(* CODESYS project Lyntupy.project
   Title: Lypuny
   Author: d2581
   Version: 0.0.0.92

Project tree, tasks and I/O mapping:
  MyController : TM241CE40T/U, Schneider Electric, order no. TM241CE40T/U, version 4.0.6.18
    application Application
      libraries: Util, 3.5.1.0 (System)
      task MAST (cyclic, interval 20 ms, priority 15, watchdog 100 ms x 1) calls FirstMastCycle, Input, PumpsFeederWater, AnalogInput, MeteoVlvPid, VlvRezervTankWtr, SetResetErr, FactorySetup, PumpsSourceWater, PumpsNetWater, Output
      global variables GVL
      global variables GVL_RETAIN
      FB/
        function block InitializationTmpGrafik [ST]
        function block OutputLimit [ST]
        function block ControlMeteoVlv [ST]
        function block ControlMeteoValve [FBD]
        function block DerjatelTemperatury [ST]
        function block OpredelaetPosition [LD]
        function block regulirovshchyk_rejyma [LD]
      PRG/
        program Input [ST]
        program Output [ST]
        program PumpsNetWater [LD]
        program PumpsFeederWater [LD]
        program PumpsSourceWater [LD]
        program VlvRezervTankWtr [LD]
        program MeteoVlvPid [FBD]
        program AnalogInput [FBD]
        program SetResetErr [LD]
        program FactorySetup [LD]
        program FirstMastCycle [CFC]
      VAR/
      global variables SystemBit
      function CheckDivDInt [ST]
      function CheckDivLInt [ST]
      function CheckDivReal [ST]
      function CheckDivLReal [ST]
    A1_IN : Digital Inputs, Schneider Electric, version 4.0.6.18
        input  idwDI_IDW0 : DWORD  // IDW0
        input  X0 : BOOL  // IDW0.I0
        input  X1 : BOOL  // IDW0.I1
        input  X2 : BOOL  // IDW0.I2
        input  X3 : BOOL  // IDW0.I3
        input  X4 : BOOL  // IDW0.I4
        input  X5 : BOOL  // IDW0.I5
        input  X6 : BOOL  // IDW0.I6
        input  X7 : BOOL  // IDW0.I7
        input  X8 : BOOL  // IDW0.I8
        input  X9 : BOOL  // IDW0.I9
        input  X10 : BOOL  // IDW0.I10
        input  X11 : BOOL  // IDW0.I11
        input  X12 : BOOL  // IDW0.I12
        input  X13 : BOOL  // IDW0.I13
        input  X14 : BOOL  // IDW0.I14
        input  X15 : BOOL  // IDW0.I15
        input  X16 : BOOL  // IDW0.I16
        input  X17 : BOOL  // IDW0.I17
        input  X18 : BOOL  // IDW0.I18
        input  X19 : BOOL  // IDW0.I19
        input  X20 : BOOL  // IDW0.I20
        input  X21 : BOOL  // IDW0.I21
        input  X22 : BOOL  // IDW0.I22
        input  X23 : BOOL  // IDW0.I23
        input  ibDI_IB1 : BYTE  // IB1
    A1_OUT : Digital Outputs, Schneider Electric, version 4.0.6.18
        output Y0 : BOOL  // QW0.Q0
        output Y1 : BOOL  // QW0.Q1
        output Y2 : BOOL  // QW0.Q2
        output Y3 : BOOL  // QW0.Q3
        output Y4 : BOOL  // QW0.Q4
        output Y5 : BOOL  // QW0.Q5
        output Y6 : BOOL  // QW0.Q6
        output Y7 : BOOL  // QW0.Q7
        output Y8 : BOOL  // QW0.Q8
        output Y9 : BOOL  // QW0.Q9
        output Y10 : BOOL  // QW0.Q10
        output Y11 : BOOL  // QW0.Q11
        output Y12 : BOOL  // QW0.Q12
        output Y13 : BOOL  // QW0.Q13
        output Y14 : BOOL  // QW0.Q14
        output Y15 : BOOL  // QW0.Q15
        output qbDQ_QB1 : BYTE  // QB1
        unmapped channels: QW0
    Counters : Counters, Schneider Electric, version 4.0.6.18
    Pulse_Generators : Pulse Generators, Schneider Electric, version 4.0.6.18
    Cartridge_1 : Cartridge, Schneider Electric, version 4.0.6.18
    Cartridge_2 : Cartridge, Schneider Electric, version 4.0.6.18
    IO_Bus : IO bus - TM3, Schneider Electric, version 4.0.6.18
      A1_1 : TM3DI16K, Schneider Electric, order no. TM3DI16K, version 1.0.1.4
          input  iwModule_1_IW0 : WORD  // IW0
          input  _1X0 : BOOL  // IW0.I0
          input  _1X1 : BOOL  // IW0.I1
          input  _1X2 : BOOL  // IW0.I2
          input  _1X3 : BOOL  // IW0.I3
          input  _1X4 : BOOL  // IW0.I4
          input  _1X5 : BOOL  // IW0.I5
          input  _1X6 : BOOL  // IW0.I6
          input  _1X7 : BOOL  // IW0.I7
          input  _1X8 : BOOL  // IW0.I8
          input  _1X9 : BOOL  // IW0.I9
          input  _1X10 : BOOL  // IW0.I10
          input  _1X11 : BOOL  // IW0.I11
          input  _1X12 : BOOL  // IW0.I12
          input  _1X13 : BOOL  // IW0.I13
          input  _1X14 : BOOL  // IW0.I14
          input  _1X15 : BOOL  // IW0.I15
      A1_2 : TM3DQ16TK, Schneider Electric, order no. TM3DQ16TK, version 1.0.1.4
          output _2Y0 : BOOL  // QW0.Q0
          output _2Y1 : BOOL  // QW0.Q1
          output _2Y2 : BOOL  // QW0.Q2
          output _2Y3 : BOOL  // QW0.Q3
          output _2Y4 : BOOL  // QW0.Q4
          output _2Y5 : BOOL  // QW0.Q5
          output _2Y6 : BOOL  // QW0.Q6
          output _2Y7 : BOOL  // QW0.Q7
          output _2Y8 : BOOL  // QW0.Q8
          output _2Y9 : BOOL  // QW0.Q9
          output _2Y10 : BOOL  // QW0.Q10
          output _2Y11 : BOOL  // QW0.Q11
          output _2Y12 : BOOL  // QW0.Q12
          output _2Y13 : BOOL  // QW0.Q13
          output _2Y14 : BOOL  // QW0.Q14
          output _2Y15 : BOOL  // QW0.Q15
          unmapped channels: QW0
      A1_3 : TM3AI4/G, Schneider Electric, order no. TM3AI4/G, version 1.0.0.15
          settings: KPI Configuration.KPI Configuration[0] = 35; KPI Configuration.KPI Configuration[1] = 35; KPI Configuration.KPI Configuration[2] = 35; KPI Configuration.KPI Configuration[3] = 35; KPI Configuration.KPI Configuration[4] = 160; KPI Configuration.KPI Configuration[5] = 15; KPI Configuration.KPI Configuration[6] = 160; KPI Configuration.KPI Configuration[7] = 15; KPI Configuration.KPI Configuration[8] = 160; KPI Configuration.KPI Configuration[9] = 15; KPI Configuration.KPI Configuration[10] = 160; KPI Configuration.KPI Configuration[11] = 15; KPI Configuration.KPI Configuration[12] = 32; KPI Configuration.KPI Configuration[13] = 78; KPI Configuration.KPI Configuration[14] = 32; KPI Configuration.KPI Configuration[15] = 78; KPI Configuration.KPI Configuration[16] = 32; KPI Configuration.KPI Configuration[17] = 78; KPI Configuration.KPI Configuration[18] = 32; KPI Configuration.KPI Configuration[19] = 78; KPI Configuration.KPI Configuration[20] = 1; KPI Configuration.KPI Configuration[22] = 1; KPI Configuration.KPI Configuration[24] = 1; KPI Configuration.KPI Configuration[26] = 1; KPI Configuration.KPI Configuration[29] = 1; KPI Configuration.KPI Configuration[30] = 1; KPI Configuration.KPI Configuration[31] = 1
          input  PE1 : INT  // IW0
          input  PE2 : INT  // IW1
          input  PE3 : INT  // IW2
          input  PERezerv : INT  // IW3
          input  ibModule_3_IBStatusIW0 : BYTE  // IBStatusIW0
          input  ibModule_3_IBStatusIW1 : BYTE  // IBStatusIW1
          input  ibModule_3_IBStatusIW2 : BYTE  // IBStatusIW2
          input  ibModule_3_IBStatusIW3 : BYTE  // IBStatusIW3
      A1_4 : TM3TI4/G, Schneider Electric, order no. TM3TI4/G, version 1.0.1.5
          settings: KPI Configuration.KPI Configuration[0] = 77; KPI Configuration.KPI Configuration[1] = 77; KPI Configuration.KPI Configuration[2] = 77; KPI Configuration.KPI Configuration[3] = 77; KPI Configuration.KPI Configuration[4] = 48; KPI Configuration.KPI Configuration[5] = 248; KPI Configuration.KPI Configuration[6] = 48; KPI Configuration.KPI Configuration[7] = 248; KPI Configuration.KPI Configuration[8] = 48; KPI Configuration.KPI Configuration[9] = 248; KPI Configuration.KPI Configuration[10] = 48; KPI Configuration.KPI Configuration[11] = 248; KPI Configuration.KPI Configuration[12] = 52; KPI Configuration.KPI Configuration[13] = 33; KPI Configuration.KPI Configuration[14] = 52; KPI Configuration.KPI Configuration[15] = 33; KPI Configuration.KPI Configuration[16] = 52; KPI Configuration.KPI Configuration[17] = 33; KPI Configuration.KPI Configuration[18] = 52; KPI Configuration.KPI Configuration[19] = 33; KPI Configuration.KPI Configuration[20] = 1; KPI Configuration.KPI Configuration[22] = 1; KPI Configuration.KPI Configuration[26] = 1
          input  TE1 : INT  // IW0
          input  TE2 : INT  // IW1
          input  TE3 : INT  // IW2
          input  TE4Rezerv : INT  // IW3
          input  ibModule_4_IBStatusIW0 : BYTE  // IBStatusIW0
          input  ibModule_4_IBStatusIW1 : BYTE  // IBStatusIW1
          input  ibModule_4_IBStatusIW2 : BYTE  // IBStatusIW2
          input  ibModule_4_IBStatusIW3 : BYTE  // IBStatusIW3
    COM_Bus : COM bus, Schneider Electric, version 4.0.6.18
    Ethernet_1 : Ethernet Network, Schneider Electric, version 4.0.6.18
        settings: IPAddress = [192, 168, 0, 32]; SubnetMask = [255, 255, 255, 0]; WebServer = TRUE; FTP Server = TRUE; SoMachine Protocol = TRUE; Modbus Server = TRUE; NetManage Protocol = TRUE; SNMP protocol = TRUE; Enable Routing = FALSE; WebVisu protocol = TRUE; DHCP Server Active = TRUE
    Serial_Line_1 : Serial line, Schneider Electric, version 4.0.6.18
      Modbus_Manager : Modbus Manager, Schneider Electric, version 4.0.0.2
    Serial_Line_2 : Serial line, Schneider Electric, version 4.0.6.18
*)

// MyController/Application/GVL
VAR_GLOBAL
	//------------------------------------------------------Inpup A1 A1.1 A1.3 A1.4-----------------------------------------
	Breake1 AT %MX0.0: BOOL;
	ErrBoiler1 AT %MX0.1: BOOL;
	ManualMode AT %MX0.2: BOOL;
	ErrBoiler2 AT %MX0.3: BOOL;
	Breake2 AT %MX0.4: BOOL;
	PressReversNetWtrLow AT %MX0.5: BOOL;
	PressReversNetWtrHigh AT %MX0.6: BOOL;
	DrySourceWtr1 AT %MX0.7: BOOL;
	WorkingPressSourceWtr1 AT %MX0.8: BOOL;
	DrySourceWtr2 AT %MX0.9: BOOL;
	WorkingPressSourceWtr2 AT %MX0.10: BOOL;
	DryNetWtr1 AT %MX0.11: BOOL;
	WorkingPressNetWtr1 AT %MX0.12: BOOL;
	DryNetWtr2 AT %MX0.13: BOOL;
	WorkingPressNetWtr2 AT %MX0.14: BOOL;
	DryFeederWtr1 AT %MX0.15: BOOL;
	WorkingPressFeederWtr1 AT %MX2.0: BOOL;
	DryFeederWtr2 AT %MX2.1: BOOL;//%MW1.1
	WorkingPressFeederWtr2 AT %MX2.2: BOOL;//%MW1.2
	PumpSourceWtr1On AT %MX2.3: BOOL;//%MW1.3
	PumpSourceWtr2On AT %MX2.4: BOOL;//%MW1.4
	PumpNetWtr1On AT %MX2.5: BOOL;//%MW1.5
	PumpNetWtr2On AT %MX2.6: BOOL;//%MW1.6
	PumpFeederWtr1On AT %MX2.7: BOOL;//%MW1.7
	PumpFeederWtr2On AT %MX2.8: BOOL;//%MW1.8
	ErrTopLevelReservTankWtr AT %MX2.9: BOOL;//%MW1.9
	TopLevelReservTankWtr AT %MX2.10: BOOL;//%MW1.10
	ErrLowLevelReservTankWtr AT %MX2.11: BOOL;//%MW1.11
	LowLevelReservTankWtr AT %MX2.12: BOOL;//%MW1.12
	Breake3 AT %MX2.13: BOOL;//%MW1.13
	// --------------------------------------------------------------резервные биты в слове -----------------------------------------------
	ErrGrafik AT %MX2.14: BOOL;
	ErrPE1 AT %MX2.15: BOOL;
	// -------------------------------------------------------------------------------------------------------------------------------------
	PressReversNetWtr AT %MD1: REAL;//%MW2,%MW3
	PressForwardNetWtr AT %MD3: REAL;//%MW6,%MW7
	PressSourceWtr AT %MD5: REAL;//%MW10,%MW11
	TpmReversNetWtr AT %MW14: INT;
	TmpAir AT %MW15: INT;
	TmpForwardWtr AT %MW16: INT;
	//------------------------------------------------------Outpun A1------------------------------------------------
	ErrPE2 AT %MX34.0: BOOL;//%MW17:X0 в панели
	PumpNetWtr1Run AT %MX34.1: BOOL;
	PumpNetWtr1Stop AT %MX34.2: BOOL;
	PumpNetWtr2Run AT %MX34.3: BOOL;
	PumpNetWtr2Stop AT %MX34.4: BOOL;
	PumpFeeder1Run AT %MX34.5: BOOL;
	PumpFeeder1Stop AT %MX34.6: BOOL;
	PumpFeeder2Run AT %MX34.7: BOOL;
	PumpFeeder2Stop AT %MX34.8: BOOL;
	PumpSourceWtr1Run AT %MX34.9: BOOL;
	PumpSourceWtr1Stop AT %MX34.10: BOOL;
	PumpSourceWtr2Run AT %MX34.11: BOOL;
	PumpSourceWtr2Stop AT %MX34.12: BOOL;
	VlvRezervTankWtrOpen AT %MX34.13: BOOL;
	RezervY13 AT %MX34.14: BOOL;
	VlvBypassOpen AT %MX34.15: BOOL;
	VlvBypassClose AT %MX36.0: BOOL;
	LightSignalColumn AT %MX36.1: BOOL;
	// --------------------------------------------------3 реле в резерве-----------------------------------------------
	Rezerv2Y1 AT %MX36.2: BOOL;
	Rezerv2Y2 AT %MX36.3: BOOL;
	Rezerv2Y3 AT %MX36.4: BOOL;
	// --------------------------------------------------резервные биты в слове-----------------------------------------
	ErrPE3 AT %MX36.5: BOOL;
	ErrTE1 AT %MX36.6: BOOL;
	ErrTE2 AT %MX36.7: BOOL;
	ErrTE3 AT %MX36.8: BOOL;
	BtnResetErr AT %MX36.9: BOOL;
	HandModeMeteo AT %MX36.10: BOOL;
	BtnRunOpnMeteoVlv AT %MX36.11: BOOL;
	BtnRunClsMeteoVlv AT %MX36.12: BOOL;
	BtnRunPumpFeederWtr1 AT %MX36.13: BOOL;
	BtnRunPumpFeederWtr2 AT %MX36.14: BOOL;
	BtnRunPumpNetWtr1 AT %MX36.15: BOOL;
	// -----------------------------------------------------------------------------------------------------------------
	BtnRunPumpNetWtr2 AT %MX80.0: BOOL;//%MW40:X0 в панели
	BtnRunPumpSourceWtr1 AT %MX80.1: BOOL;
	BtnRunPumpSourceWtr2 AT %MX80.2: BOOL;
	BtnVlvRezervTankWtrOpen AT %MX80.3: BOOL;//%MW40:X3
	ErrAll AT %MX80.4: BOOL;//%MW40:X4
	BtnSetFactorySetup AT %MX80.5: BOOL;//%MW40:X5
	bool6 AT %MX80.6: BOOL;//%MW40:X6
	bool7 AT %MX80.7: BOOL;//%MW40:X7
	bool8 AT %MX80.8: BOOL;//%MW40:X8
	bool9 AT %MX80.9: BOOL;//%MW40:X9
	bool10 AT %MX80.10: BOOL;//%MW40:X10
	bool11 AT %MX80.11: BOOL;//%MW40:X11
	bool12 AT %MX80.12: BOOL;//%MW40:X12
	bool13 AT %MX80.13: BOOL;//%MW40:X13
	bool14 AT %MX80.14: BOOL;//%MW40:X14
	bool15 AT %MX80.15: BOOL;//%MW40:X15
	
	LevelRezervTankWtr AT %MW41: INT;
	ZadanieForMeteoVlv AT %MW42: INT;

END_VAR

// MyController/Application/GVL_RETAIN
VAR_GLOBAL RETAIN
	PE1Min AT %MW4: INT;
	PE1Max AT %MW5: INT;
	PE2Min AT %MW8: INT;
	PE2Max AT %MW9: INT;
	PE3Min AT %MW12: INT;
	PE3Max AT %MW13: INT;
	
	
	TmpGrafN22 AT %MW19: WORD;
	TmpGrafN19 AT %MW20: WORD;
	TmpGrafN15 AT %MW21: WORD;
	TmpGrafN13 AT %MW22: WORD;
	TmpGrafN10 AT %MW23: WORD;
	TmpGrafN7 AT %MW24: WORD;
	TmpGrafN3 AT %MW25: WORD;
	TmpGrafP0 AT %MW26: WORD;
	TmpGrafP2 AT %MW27: WORD;
	TmpGrafP5 AT %MW28: WORD;
	TmpgrafP10 AT %MW29: WORD;
	
	KL: ARRAY[0..10] OF POINT;
	
	KpVlv AT %MD15: REAL;// %MW30, %MW31
	TnVlv AT %MD16: REAL;// %MW32, %MW33
	TvVlv AT %MD17: REAL;// %MW34, %MW35
	MaxVlv AT %MW36: INT;//Максимальная величина открытия задвижки в %
	MinVlv AT %MW37: INT;//Минимальная величина закрытия задвижки в %
	TimeMoveVlv AT %MW38: INT;//Время открытия задвижки в секундах
	CurrentPositionVlv AT %MW39: INT;// Текущее положение
	
	UseM1 AT %MX86.0: BOOL;
	UseM2 AT %MX86.1: BOOL;
	UseM3 AT %MX86.2: BOOL;
	UseM4 AT %MX86.3: BOOL;
	UseM5 AT %MX86.4: BOOL;
	UseM6 AT %MX86.5: BOOL;
	
	CurrentPosition: INT;
END_VAR

// MyController/Application/SystemBit
VAR_GLOBAL
	// Indicates or executes a cold start (data initialized to default values)
	SB_COLDSTART: BOOL;
	// Indicates there was a warm start with data backup
	SB_WARMSTART: BOOL;
	// Time base of 1 min generated by an internal clock
	SB_TB1MIN: BOOL;
	// Time base of 1 sek generated by an internal clock
	SB_TB1SEK: BOOL;
	// Indicates the first controller cycle in RUN mode
	SB_FIRSTRUN: BOOL;
END_VAR

// MyController/Application/PRG/FirstMastCycle
PROGRAM FirstMastCycle
VAR
	tm_firstrun: TOF;
	BLINK_1sek: Util.BLINK;
END_VAR
VAR // added by the converter: edge detectors and wires of the graphical bodies
    _w1 : ANY;
END_VAR

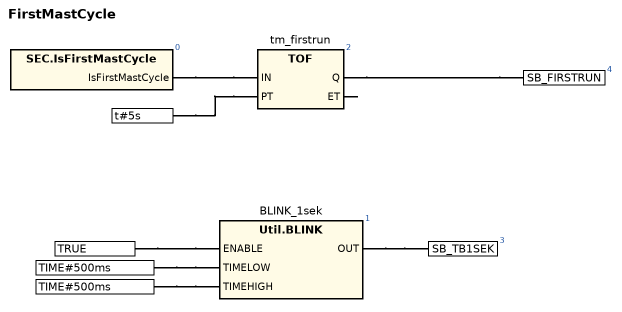
_w1 := SEC.IsFirstMastCycle();
BLINK_1sek(ENABLE := TRUE, TIMELOW := TIME#500ms, TIMEHIGH := TIME#500ms); // Util.BLINK
tm_firstrun(IN := _w1, PT := t#5s); // TOF
SB_TB1SEK := BLINK_1sek.OUT;
SB_FIRSTRUN := tm_firstrun.Q;

END_PROGRAM

// MyController/Application/PRG/Input
PROGRAM Input
VAR
END_VAR

Breake1 := 	NOT X0;
ErrBoiler1 := X1;
ManualMode := X2;
ErrBoiler2 := X3;
Breake2 := X4;
PressReversNetWtrLow := NOT X5;//PIS9
PressReversNetWtrHigh := NOT X6;//PIS9
DrySourceWtr1 := NOT X7;//PIS7
WorkingPressSourceWtr1:= NOT X8;//PIS5
DrySourceWtr2 := NOT X9;//PIS8
WorkingPressSourceWtr2 := NOT X10;//PIS6
DryNetWtr1 := NOT X11;//PIS3
WorkingPressNetWtr1 := NOT X12;//PIS1
DryNetWtr2 := NOT X13;//PIS4
WorkingPressNetWtr2 := NOT X14;//PIS2
DryFeederWtr1 := NOT X15;//PIS11
WorkingPressFeederWtr1 := NOT X16; //PIS9
DryFeederWtr2 := NOT X17;//PIS12
WorkingPressFeederWtr2 := NOT X18; //PIS12
PumpSourceWtr1On := X19;//KM-K6.1
PumpSourceWtr2On := X20;//KM-K6.2
PumpNetWtr1On := X21;//KM-K3.1
PumpNetWtr2On := X22;//KM-K3.2
PumpFeederWtr1On :=	X23;//KM-K4.1
PumpFeederWtr2On := _1X0;//KM-K4.2
ErrTopLevelReservTankWtr := _1X4;//Верхний аварийный уровень в баке запаса воды
TopLevelReservTankWtr := _1X3;//Верхний рабочий уровень в баке запаса воды
ErrLowLevelReservTankWtr := _1X1;//Нижний аварийный уровень в баке запаса воды
LowLevelReservTankWtr := _1X2;//Нижний рабочий уровень в баке запаса воды
Breake3 := _1X5;

PressReversNetWtr := AnalogInput.LinTrafoPressReversNetWtr.OUT;//Давление обратной сетевой воды
PressForwardNetWtr := AnalogInput.LinTrafoPressForwardNetWtr.OUT;//Давление прямой сетевой воды 
PressSourceWtr := AnalogInput.LinTrafoPressSourceWtr.OUT;;//Давление исходной сетевой воды 

TpmReversNetWtr := TE1;//Температура обратной сетевой воды на входе в котельную
TmpForwardWtr := TE2;//Температура прямой сетевой воды на выходе из котельной
TmpAir := TE3;//Температура наружнего воздуха

END_PROGRAM

// MyController/Application/PRG/AnalogInput
PROGRAM AnalogInput
VAR
	LinTrafoPressReversNetWtr: LIN_TRAFO;
	LinTrafoPressForwardNetWtr: LIN_TRAFO;
	LinTrafoPressSourceWtr: LIN_TRAFO;
	ErrPE1: BOOL;
	ErrPE2: BOOL;
	ErrPE3: BOOL;
END_VAR

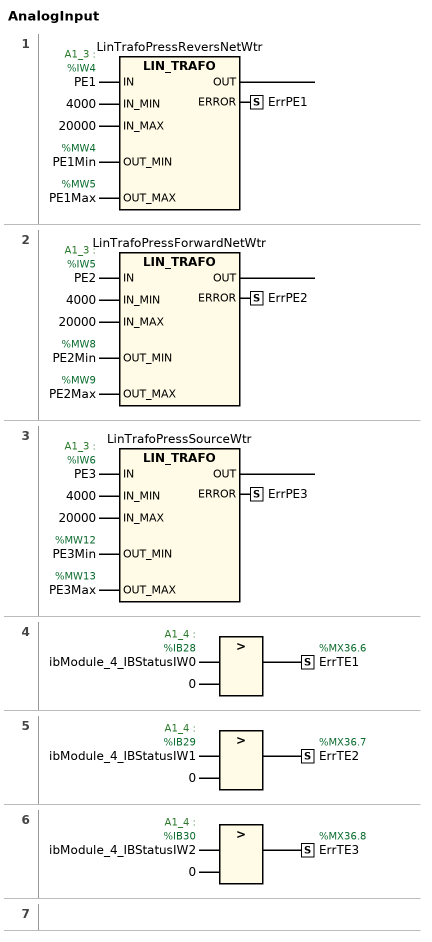
// NETWORK 1
//   PE1: A1_3 : | AT %IW4
//   PE1Min: AT %MW4
//   PE1Max: AT %MW5
LinTrafoPressReversNetWtr(IN := PE1, IN_MIN := 4000, IN_MAX := 20000, OUT_MIN := PE1Min, OUT_MAX := PE1Max); // LIN_TRAFO
ErrPE1 S= LinTrafoPressReversNetWtr.ERROR;

// NETWORK 2
//   PE2: A1_3 : | AT %IW5
//   PE2Min: AT %MW8
//   PE2Max: AT %MW9
LinTrafoPressForwardNetWtr(IN := PE2, IN_MIN := 4000, IN_MAX := 20000, OUT_MIN := PE2Min, OUT_MAX := PE2Max); // LIN_TRAFO
ErrPE2 S= LinTrafoPressForwardNetWtr.ERROR;

// NETWORK 3
//   PE3: A1_3 : | AT %IW6
//   PE3Min: AT %MW12
//   PE3Max: AT %MW13
LinTrafoPressSourceWtr(IN := PE3, IN_MIN := 4000, IN_MAX := 20000, OUT_MIN := PE3Min, OUT_MAX := PE3Max); // LIN_TRAFO
ErrPE3 S= LinTrafoPressSourceWtr.ERROR;

// NETWORK 4
//   ibModule_4_IBStatusIW0: A1_4 : | AT %IB28
//   ErrTE1: AT %MX36.6
ErrTE1 S= ibModule_4_IBStatusIW0 > 0;

// NETWORK 5
//   ibModule_4_IBStatusIW1: A1_4 : | AT %IB29
//   ErrTE2: AT %MX36.7
ErrTE2 S= ibModule_4_IBStatusIW1 > 0;

// NETWORK 6
//   ibModule_4_IBStatusIW2: A1_4 : | AT %IB30
//   ErrTE3: AT %MX36.8
ErrTE3 S= ibModule_4_IBStatusIW2 > 0;

// NETWORK 7

END_PROGRAM

// MyController/Application/PRG/PumpsFeederWater
PROGRAM PumpsFeederWater
VAR
	PulsRunPumpFeederWtr1: TP;
	PulsStopPumpFeederWtr1: TP;
	PulsStopPumpFeederWtr2: TP;
	PulsRunPumpFeederWtr2: TP;
END_VAR
VAR // added by the converter: edge detectors and wires of the graphical bodies
    _w1 : BOOL;
    _rt1, _rt2, _rt3, _rt4 : R_TRIG;
    _ft1, _ft2 : F_TRIG;
END_VAR

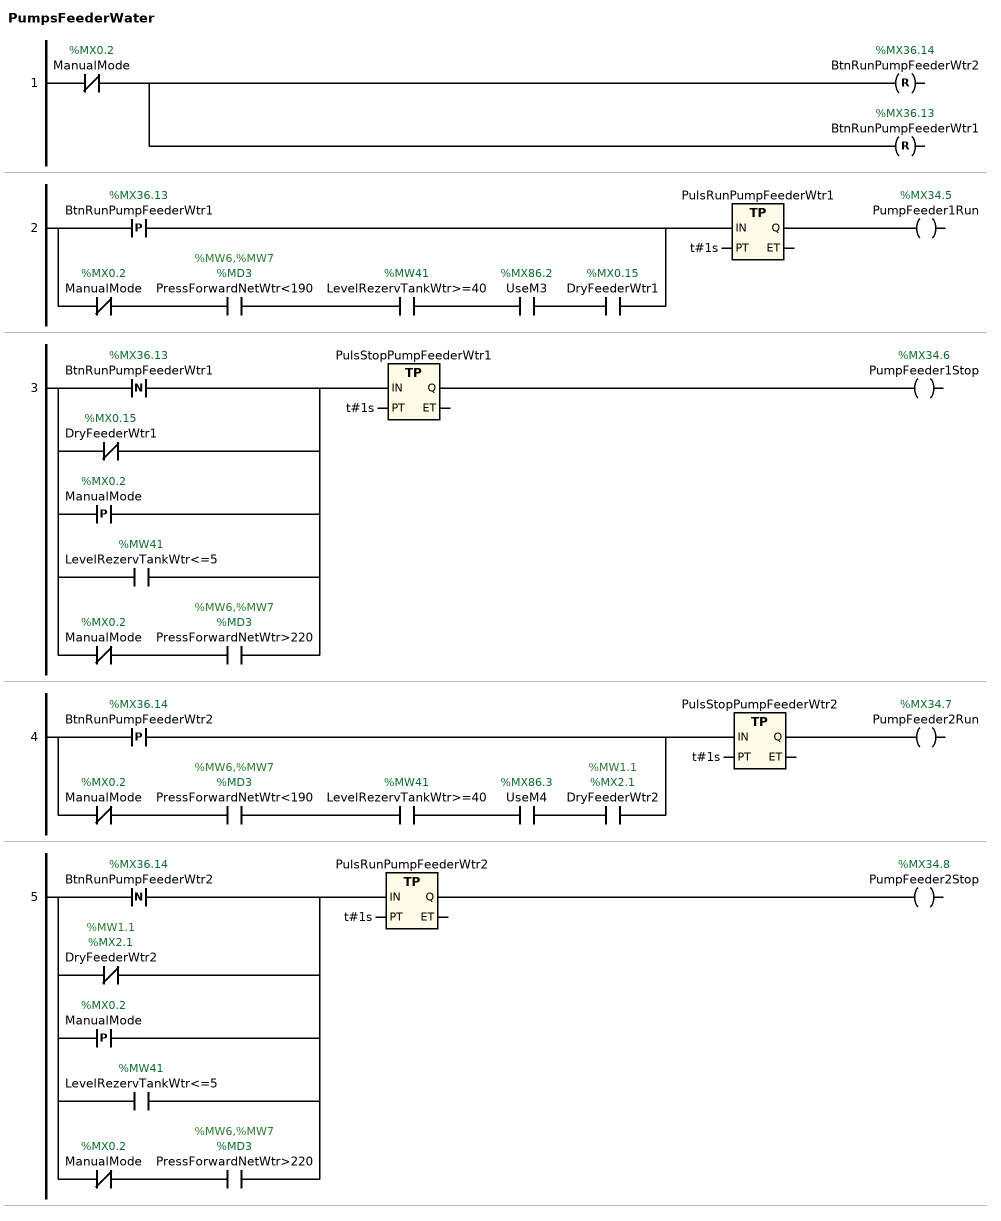
// NETWORK 1
//   ManualMode: AT %MX0.2
//   BtnRunPumpFeederWtr2: AT %MX36.14
//   BtnRunPumpFeederWtr1: AT %MX36.13
_w1 := NOT ManualMode;
BtnRunPumpFeederWtr2 R= _w1;
BtnRunPumpFeederWtr1 R= _w1;

// NETWORK 2
//   BtnRunPumpFeederWtr1: AT %MX36.13
//   ManualMode: AT %MX0.2
//   PressForwardNetWtr<190: %MW6,%MW7 | AT %MD3
//   LevelRezervTankWtr>=40: AT %MW41
//   UseM3: AT %MX86.2
//   DryFeederWtr1: AT %MX0.15
//   PumpFeeder1Run: AT %MX34.5
_rt1(CLK := BtnRunPumpFeederWtr1);
PulsRunPumpFeederWtr1(IN := _rt1.Q OR (NOT ManualMode AND (PressForwardNetWtr<190) AND (LevelRezervTankWtr>=40)) AND UseM3 AND DryFeederWtr1, PT := t#1s); // TP
PumpFeeder1Run := PulsRunPumpFeederWtr1.Q;

// NETWORK 3
//   BtnRunPumpFeederWtr1: AT %MX36.13
//   DryFeederWtr1: AT %MX0.15
//   ManualMode: AT %MX0.2
//   LevelRezervTankWtr<=5: AT %MW41
//   PressForwardNetWtr>220: %MW6,%MW7 | AT %MD3
//   PumpFeeder1Stop: AT %MX34.6
_ft1(CLK := BtnRunPumpFeederWtr1);
_rt2(CLK := ManualMode);
PulsStopPumpFeederWtr1(IN := _ft1.Q OR NOT DryFeederWtr1 OR (_rt2.Q OR (LevelRezervTankWtr<=5)) OR NOT ManualMode AND (PressForwardNetWtr>220), PT := t#1s); // TP
PumpFeeder1Stop := PulsStopPumpFeederWtr1.Q;

// NETWORK 4
//   BtnRunPumpFeederWtr2: AT %MX36.14
//   ManualMode: AT %MX0.2
//   PressForwardNetWtr<190: %MW6,%MW7 | AT %MD3
//   LevelRezervTankWtr>=40: AT %MW41
//   UseM4: AT %MX86.3
//   DryFeederWtr2: %MW1.1 | AT %MX2.1
//   PumpFeeder2Run: AT %MX34.7
_rt3(CLK := BtnRunPumpFeederWtr2);
PulsStopPumpFeederWtr2(IN := _rt3.Q OR (NOT ManualMode AND (PressForwardNetWtr<190) AND (LevelRezervTankWtr>=40)) AND UseM4 AND DryFeederWtr2, PT := t#1s); // TP
PumpFeeder2Run := PulsStopPumpFeederWtr2.Q;

// NETWORK 5
//   BtnRunPumpFeederWtr2: AT %MX36.14
//   DryFeederWtr2: %MW1.1 | AT %MX2.1
//   ManualMode: AT %MX0.2
//   LevelRezervTankWtr<=5: AT %MW41
//   PressForwardNetWtr>220: %MW6,%MW7 | AT %MD3
//   PumpFeeder2Stop: AT %MX34.8
_ft2(CLK := BtnRunPumpFeederWtr2);
_rt4(CLK := ManualMode);
PulsRunPumpFeederWtr2(IN := _ft2.Q OR NOT DryFeederWtr2 OR (_rt4.Q OR (LevelRezervTankWtr<=5)) OR NOT ManualMode AND (PressForwardNetWtr>220), PT := t#1s); // TP
PumpFeeder2Stop := PulsRunPumpFeederWtr2.Q;

END_PROGRAM

// MyController/Application/PRG/MeteoVlvPid
PROGRAM MeteoVlvPid
VAR
	GraficPodachi: CHARCURVE;
	OutputLimit_TmpAir: OutputLimit;
	InitializationTmpGrafik_Podachy: InitializationTmpGrafik;
	PID_Valve: PID;
	
	ControlMeteoVlvNetWtr: ControlMeteoValve;
	DerjatelTemperatury_0: DerjatelTemperatury;
	positionVlv: OpredelaetPosition;
	manual_auto: regulirovshchyk_rejyma;
END_VAR

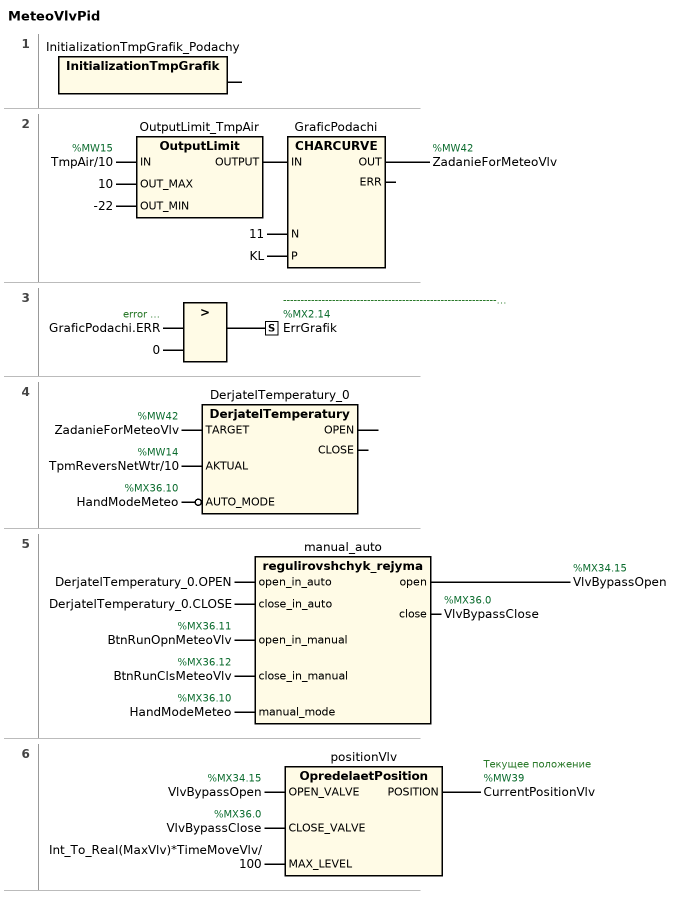
// NETWORK 1
InitializationTmpGrafik_Podachy(); // InitializationTmpGrafik

// NETWORK 2
//   TmpAir/10: AT %MW15
//   ZadanieForMeteoVlv: AT %MW42
OutputLimit_TmpAir(IN := TmpAir/10, OUT_MAX := 10, OUT_MIN := -22); // OutputLimit
GraficPodachi(IN := OutputLimit_TmpAir.OUTPUT, N := 11, P := KL); // CHARCURVE
ZadanieForMeteoVlv := GraficPodachi.OUT;

// NETWORK 3
//   GraficPodachi.ERR: error : 0 : no error 1 : error in ARRAY: wrong sequence ( completely tested, only if IN is equal to largest X-value of P) 2 : IN outside of limits of P 4 : number of POINTS (N) invalid
//   ErrGrafik: --------------------------------------------------------------резервные биты в слове ----------------------------------------------- | AT %MX2.14
ErrGrafik S= GraficPodachi.ERR > 0;

// NETWORK 4
//   ZadanieForMeteoVlv: AT %MW42
//   TpmReversNetWtr/10: AT %MW14
//   HandModeMeteo: AT %MX36.10
DerjatelTemperatury_0(
    TARGET := ZadanieForMeteoVlv,
    AKTUAL := TpmReversNetWtr/10,
    AUTO_MODE := NOT HandModeMeteo); // DerjatelTemperatury

// NETWORK 5
//   BtnRunOpnMeteoVlv: AT %MX36.11
//   BtnRunClsMeteoVlv: AT %MX36.12
//   HandModeMeteo: AT %MX36.10
//   VlvBypassClose: AT %MX36.0
//   VlvBypassOpen: AT %MX34.15
manual_auto(
    open_in_auto := DerjatelTemperatury_0.OPEN,
    close_in_auto := DerjatelTemperatury_0.CLOSE,
    open_in_manual := BtnRunOpnMeteoVlv,
    close_in_manual := BtnRunClsMeteoVlv,
    manual_mode := HandModeMeteo,
    close => VlvBypassClose); // regulirovshchyk_rejyma
VlvBypassOpen := manual_auto.open;

// NETWORK 6
//   VlvBypassOpen: AT %MX34.15
//   VlvBypassClose: AT %MX36.0
//   CurrentPositionVlv: Текущее положение | AT %MW39
positionVlv(
    OPEN_VALVE := VlvBypassOpen,
    CLOSE_VALVE := VlvBypassClose,
    MAX_LEVEL := Int_To_Real(MaxVlv)*TimeMoveVlv/100); // OpredelaetPosition
CurrentPositionVlv := positionVlv.POSITION;

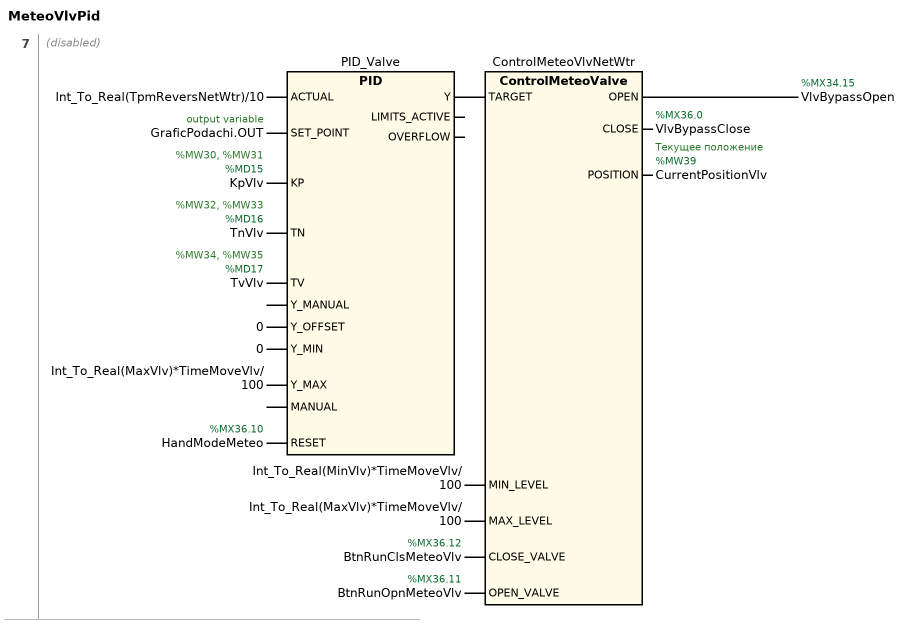
// NETWORK 7 (disabled)
//   GraficPodachi.OUT: output variable
//   KpVlv: %MW30, %MW31 | AT %MD15
//   TnVlv: %MW32, %MW33 | AT %MD16
//   TvVlv: %MW34, %MW35 | AT %MD17
//   HandModeMeteo: AT %MX36.10
//   BtnRunClsMeteoVlv: AT %MX36.12
//   BtnRunOpnMeteoVlv: AT %MX36.11
//   VlvBypassClose: AT %MX36.0
//   CurrentPositionVlv: Текущее положение | AT %MW39
//   VlvBypassOpen: AT %MX34.15
// PID_Valve(
//     ACTUAL := Int_To_Real(TpmReversNetWtr)/10,
//     SET_POINT := GraficPodachi.OUT,
//     KP := KpVlv,
//     TN := TnVlv,
//     TV := TvVlv,
//     Y_OFFSET := 0,
//     Y_MIN := 0,
//     Y_MAX := Int_To_Real(MaxVlv)*TimeMoveVlv/100,
//     RESET := HandModeMeteo); // PID
// ControlMeteoVlvNetWtr(
//     TARGET := PID_Valve.Y,
//     MIN_LEVEL := Int_To_Real(MinVlv)*TimeMoveVlv/100,
//     MAX_LEVEL := Int_To_Real(MaxVlv)*TimeMoveVlv/100,
//     CLOSE_VALVE := BtnRunClsMeteoVlv,
//     OPEN_VALVE := BtnRunOpnMeteoVlv,
//     CLOSE => VlvBypassClose,
//     POSITION => CurrentPositionVlv); // ControlMeteoValve
// VlvBypassOpen := ControlMeteoVlvNetWtr.OPEN;

END_PROGRAM

// MyController/Application/FB/InitializationTmpGrafik
FUNCTION_BLOCK InitializationTmpGrafik
VAR_INPUT
END_VAR
VAR_OUTPUT
END_VAR
VAR
END_VAR

KL[0].X:=-22;KL[0].Y:=TmpGrafN22;
KL[1].X:=-19;KL[1].Y:=TmpGrafN19;
KL[2].X:=-15;KL[2].Y:=TmpGrafN15;
KL[3].X:=-13;KL[3].Y:=TmpGrafN13;
KL[4].X:=-10;KL[4].Y:=TmpGrafN10;
KL[5].X:=-7;KL[5].Y:=TmpGrafN7;
KL[6].X:=-3;KL[6].Y:=TmpGrafN3;
KL[7].X:=0;KL[7].Y:=TmpGrafP0;
KL[8].X:=2;KL[8].Y:=TmpGrafP2;
KL[9].X:=5;KL[9].Y:=TmpGrafP5;
KL[10].X:=10;KL[10].Y:=TmpGrafP10;

END_FUNCTION_BLOCK

// MyController/Application/FB/OutputLimit
FUNCTION_BLOCK OutputLimit
VAR_INPUT
	IN: INT;
	OUT_MAX: INT;
	OUT_MIN: INT;
END_VAR
VAR_OUTPUT
	OUTPUT: INT;
END_VAR
VAR
END_VAR

IF	IN>OUT_MAX THEN OUTPUT:=OUT_MAX;
ELSIF IN<OUT_MIN THEN OUTPUT:=OUT_MIN;
ELSE OUTPUT:=IN;
END_IF

END_FUNCTION_BLOCK

// MyController/Application/PRG/Output
PROGRAM Output
VAR	
END_VAR

IF NOT SB_FIRSTRUN THEN
	Y0 := PumpNetWtr1Run;
	Y1 := PumpNetWtr1Stop;
	Y2 := PumpNetWtr2Run;
	Y3 := PumpNetWtr2Stop;
	Y4 := PumpFeeder1Run;
	Y5 := PumpFeeder1Stop;
	Y6 :=  PumpFeeder2Run;
	Y7 := PumpFeeder2Stop;
	Y8 := PumpSourceWtr1Run;
	Y9 := PumpSourceWtr1Stop;
	Y10 := PumpSourceWtr2Run;
	Y11 := PumpSourceWtr2Stop;
	Y12 := VlvRezervTankWtrOpen;
	Y13 := RezervY13;
	Y14 := VlvBypassClose; 
	Y15 :=VlvBypassOpen;
	_2Y0 := LightSignalColumn;
	_2Y1 := Rezerv2Y1;
	_2Y2 := Rezerv2Y2;
	_2Y3 := Rezerv2Y3;	
END_IF

END_PROGRAM

// MyController/Application/FB/DerjatelTemperatury
FUNCTION_BLOCK DerjatelTemperatury
VAR_INPUT
	TARGET: INT;
	AKTUAL: INT;
	AUTO_MODE: BOOL;
END_VAR
VAR_OUTPUT
	OPEN: BOOL;
	CLOSE: BOOL;
END_VAR
VAR
	oshibka: INT;
	tm_Low_5s_Hi_1s: BLINK;
	to_open: BOOL;
	to_close: BOOL;
END_VAR

oshibka:=TARGET-AKTUAL;

tm_Low_5s_hi_1s(ENABLE:=(to_open OR to_close OR tm_Low_5s_hi_1s.OUT), TIMELOW:=T#10S, TIMEHIGH:=T#1S);//Запускаем моргалку для медленного перемещения задвижки

IF oshibka>1 THEN
	to_open:=TRUE;
	to_close:=FALSE;
ELSE 
	to_open:=FALSE;
END_IF
IF oshibka<-1 THEN
	to_open:=FALSE;
	to_close:=TRUE;
ELSE
	to_close:=FALSE;
END_IF

IF AUTO_MODE THEN
 	OPEN:=to_open AND tm_Low_5s_hi_1s.OUT;// подаем сигнал на выход модулируя его моргалкой
	CLOSE:=to_close AND tm_Low_5s_hi_1s.OUT;
END_IF

END_FUNCTION_BLOCK

// MyController/Application/FB/regulirovshchyk_rejyma
// Направляет сигнал на выход с кнопок или с регулятора температуры
FUNCTION_BLOCK regulirovshchyk_rejyma 
VAR_INPUT
	open_in_auto: BOOL;
	close_in_auto: BOOL;
	open_in_manual: BOOL;
	close_in_manual: BOOL;
	manual_mode: BOOL;
END_VAR
VAR_OUTPUT
	open: BOOL;
	close: BOOL;
END_VAR
VAR
END_VAR

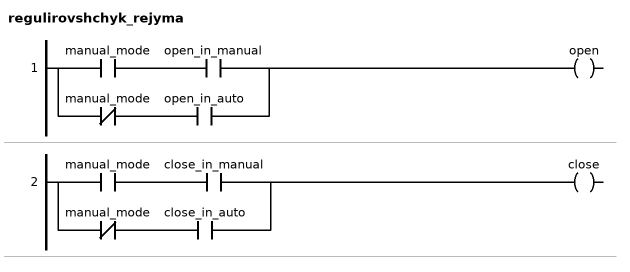
// NETWORK 1
open := manual_mode AND open_in_manual OR NOT manual_mode AND open_in_auto;

// NETWORK 2
close := manual_mode AND close_in_manual OR NOT manual_mode AND close_in_auto;

END_FUNCTION_BLOCK

// MyController/Application/FB/OpredelaetPosition
//Рассчитывает количество секунд которые в течении которых 
//на входе был сигнал и переводит их в проценты открытия
FUNCTION_BLOCK OpredelaetPosition
VAR_INPUT
	OPEN_VALVE: BOOL;
	CLOSE_VALVE: BOOL;
	MAX_LEVEL: REAL;
	
END_VAR
VAR_OUTPUT
	POSITION: INT;
END_VAR
VAR
	OutputLimitPOSITION1: OutputLimit;
	blink2_1sek: BLINK;
	blink1_1sek: BLINK;
	//CurrentPosition: INT; я эту переменную перенес в GLOBAL_RETAIN	
END_VAR
VAR // added by the converter: edge detectors and wires of the graphical bodies
    _rt1, _rt2 : R_TRIG;
END_VAR

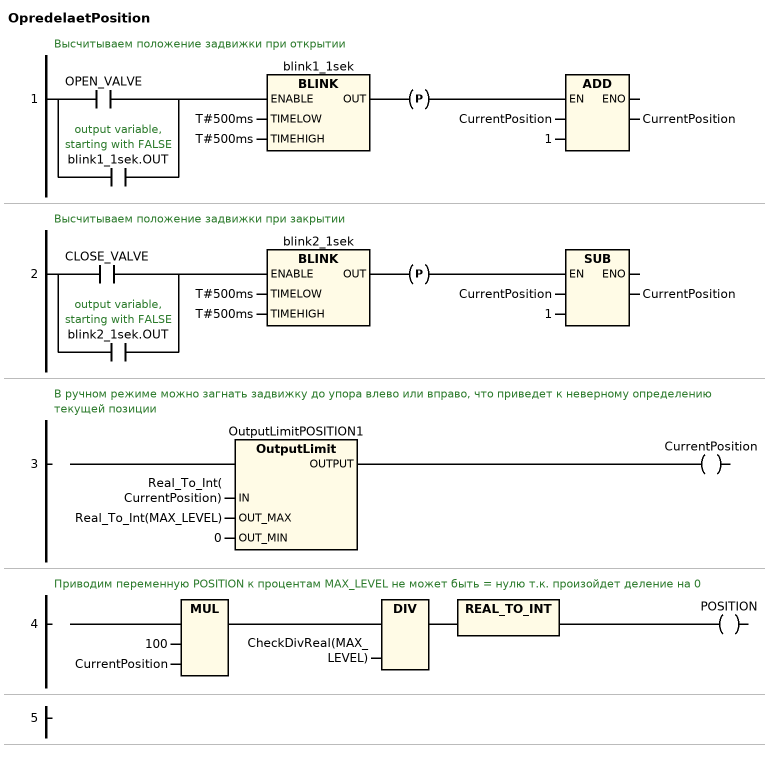
// NETWORK 1
// Высчитываем положение задвижки при открытии
//   blink1_1sek.OUT: output variable, starting with FALSE
blink1_1sek(ENABLE := OPEN_VALVE OR blink1_1sek.OUT, TIMELOW := T#500ms, TIMEHIGH := T#500ms); // BLINK
_rt1(CLK := blink1_1sek.OUT);
IF _rt1.Q THEN CurrentPosition := CurrentPosition + 1; END_IF

// NETWORK 2
// Высчитываем положение задвижки при закрытии
//   blink2_1sek.OUT: output variable, starting with FALSE
blink2_1sek(ENABLE := CLOSE_VALVE OR blink2_1sek.OUT, TIMELOW := T#500ms, TIMEHIGH := T#500ms); // BLINK
_rt2(CLK := blink2_1sek.OUT);
IF _rt2.Q THEN CurrentPosition := CurrentPosition - 1; END_IF

// NETWORK 3
// В ручном режиме можно загнать задвижку до упора влево или вправо, что приведет к неверному определению текущей позиции
OutputLimitPOSITION1(IN := Real_To_Int(CurrentPosition), OUT_MAX := Real_To_Int(MAX_LEVEL), OUT_MIN := 0); // OutputLimit
CurrentPosition := OutputLimitPOSITION1.OUTPUT;

// NETWORK 4
// Приводим переменную POSITION к процентам MAX_LEVEL не может быть = нулю т.к. произойдет деление на 0
POSITION := REAL_TO_INT((100 * CurrentPosition) / (CheckDivReal(MAX_LEVEL)));

// NETWORK 5

END_FUNCTION_BLOCK

// MyController/Application/CheckDivReal
// Implicitly generated code : DO NOT EDIT
FUNCTION CheckDivReal : REAL
VAR_INPUT
	divisor:REAL;
END_VAR

// Implicitly generated code : Only an Implementation suggestion
IF divisor = 0 THEN
	CheckDivReal:=1;
ELSE
	CheckDivReal:=divisor;
END_IF;

END_FUNCTION

// MyController/Application/FB/ControlMeteoValve
FUNCTION_BLOCK ControlMeteoValve
VAR_INPUT
	TARGET: REAL;
	MIN_LEVEL: REAL;
	MAX_LEVEL: REAL;
	CLOSE_VALVE: BOOL;
	OPEN_VALVE: BOOL;
	
END_VAR
VAR_OUTPUT
	OPEN: BOOL;
	CLOSE: BOOL;
	POSITION: INT;
END_VAR
VAR
	PulsValveOpn: BLINK;
	PulsValveCls: BLINK;
	blink1_1s: BLINK;
	blink2_1s: BLINK;
	CurrentPosition: INT;
	OutputLimitPOSITION: OutputLimit;
END_VAR
VAR // added by the converter: edge detectors and wires of the graphical bodies
    _rt1, _rt2, _rt3, _rt4 : R_TRIG;
END_VAR

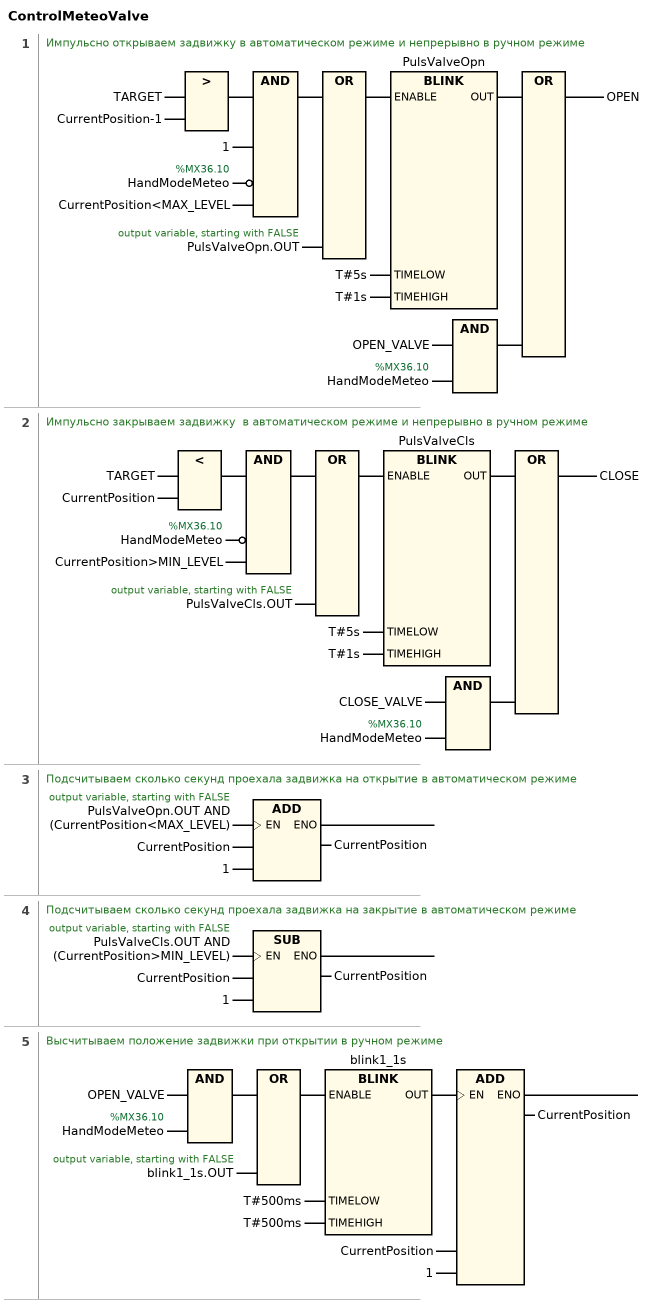
// NETWORK 1
// Импульсно открываем задвижку в автоматическом режиме и непрерывно в ручном режиме
//   HandModeMeteo: AT %MX36.10
//   PulsValveOpn.OUT: output variable, starting with FALSE
PulsValveOpn(
    ENABLE := TARGET > (CurrentPosition-1) AND 1 AND NOT HandModeMeteo AND (CurrentPosition<MAX_LEVEL) OR PulsValveOpn.OUT,
    TIMELOW := T#5s,
    TIMEHIGH := T#1s); // BLINK
OPEN := PulsValveOpn.OUT OR OPEN_VALVE AND HandModeMeteo;

// NETWORK 2
// Импульсно закрываем задвижку  в автоматическом режиме и непрерывно в ручном режиме
//   HandModeMeteo: AT %MX36.10
//   PulsValveCls.OUT: output variable, starting with FALSE
PulsValveCls(
    ENABLE := TARGET < CurrentPosition AND NOT HandModeMeteo AND (CurrentPosition>MIN_LEVEL) OR PulsValveCls.OUT,
    TIMELOW := T#5s,
    TIMEHIGH := T#1s); // BLINK
CLOSE := PulsValveCls.OUT OR CLOSE_VALVE AND HandModeMeteo;

// NETWORK 3
// Подсчитываем сколько секунд проехала задвижка на открытие в автоматическом режиме
//   PulsValveOpn.OUT AND (CurrentPosition<MAX_LEVEL): output variable, starting with FALSE
_rt1(CLK := PulsValveOpn.OUT AND (CurrentPosition<MAX_LEVEL));
IF _rt1.Q THEN CurrentPosition := CurrentPosition + 1; END_IF

// NETWORK 4
// Подсчитываем сколько секунд проехала задвижка на закрытие в автоматическом режиме
//   PulsValveCls.OUT AND (CurrentPosition>MIN_LEVEL): output variable, starting with FALSE
_rt2(CLK := PulsValveCls.OUT AND (CurrentPosition>MIN_LEVEL));
IF _rt2.Q THEN CurrentPosition := CurrentPosition - 1; END_IF

// NETWORK 5
// Высчитываем положение задвижки при открытии в ручном режиме
//   HandModeMeteo: AT %MX36.10
//   blink1_1s.OUT: output variable, starting with FALSE
blink1_1s(ENABLE := OPEN_VALVE AND HandModeMeteo OR blink1_1s.OUT, TIMELOW := T#500ms, TIMEHIGH := T#500ms); // BLINK
_rt3(CLK := blink1_1s.OUT);
IF _rt3.Q THEN CurrentPosition := CurrentPosition + 1; END_IF

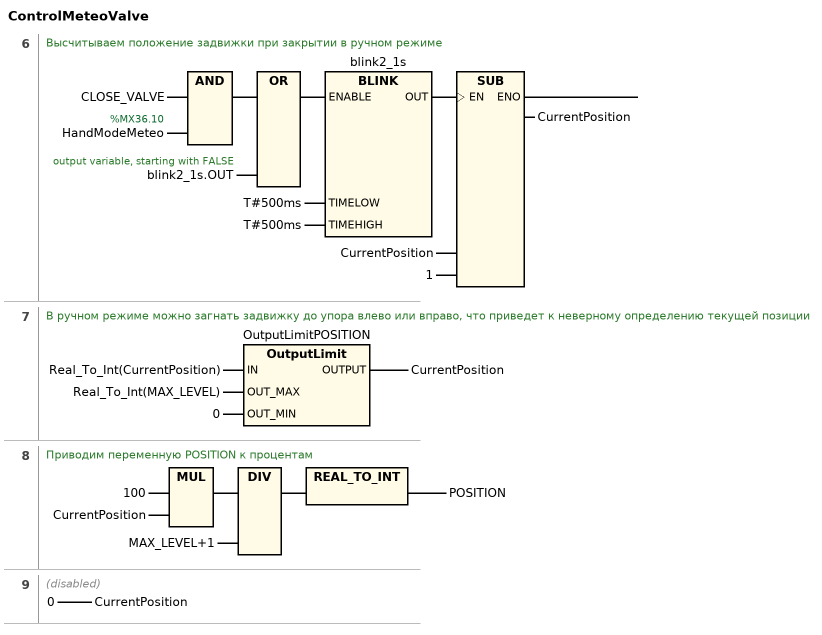
// NETWORK 6
// Высчитываем положение задвижки при закрытии в ручном режиме
//   HandModeMeteo: AT %MX36.10
//   blink2_1s.OUT: output variable, starting with FALSE
blink2_1s(ENABLE := CLOSE_VALVE AND HandModeMeteo OR blink2_1s.OUT, TIMELOW := T#500ms, TIMEHIGH := T#500ms); // BLINK
_rt4(CLK := blink2_1s.OUT);
IF _rt4.Q THEN CurrentPosition := CurrentPosition - 1; END_IF

// NETWORK 7
// В ручном режиме можно загнать задвижку до упора влево или вправо, что приведет к неверному определению текущей позиции
OutputLimitPOSITION(IN := Real_To_Int(CurrentPosition), OUT_MAX := Real_To_Int(MAX_LEVEL), OUT_MIN := 0); // OutputLimit
CurrentPosition := OutputLimitPOSITION.OUTPUT;

// NETWORK 8
// Приводим переменную POSITION к процентам
POSITION := REAL_TO_INT((100 * CurrentPosition) / (MAX_LEVEL+1));

// NETWORK 9 (disabled)
// CurrentPosition := 0;

END_FUNCTION_BLOCK

// MyController/Application/PRG/VlvRezervTankWtr
PROGRAM VlvRezervTankWtr
VAR
END_VAR
VAR // added by the converter: edge detectors and wires of the graphical bodies
    _rt1 : R_TRIG;
    _ft1 : F_TRIG;
    _w1 : BOOL;
END_VAR

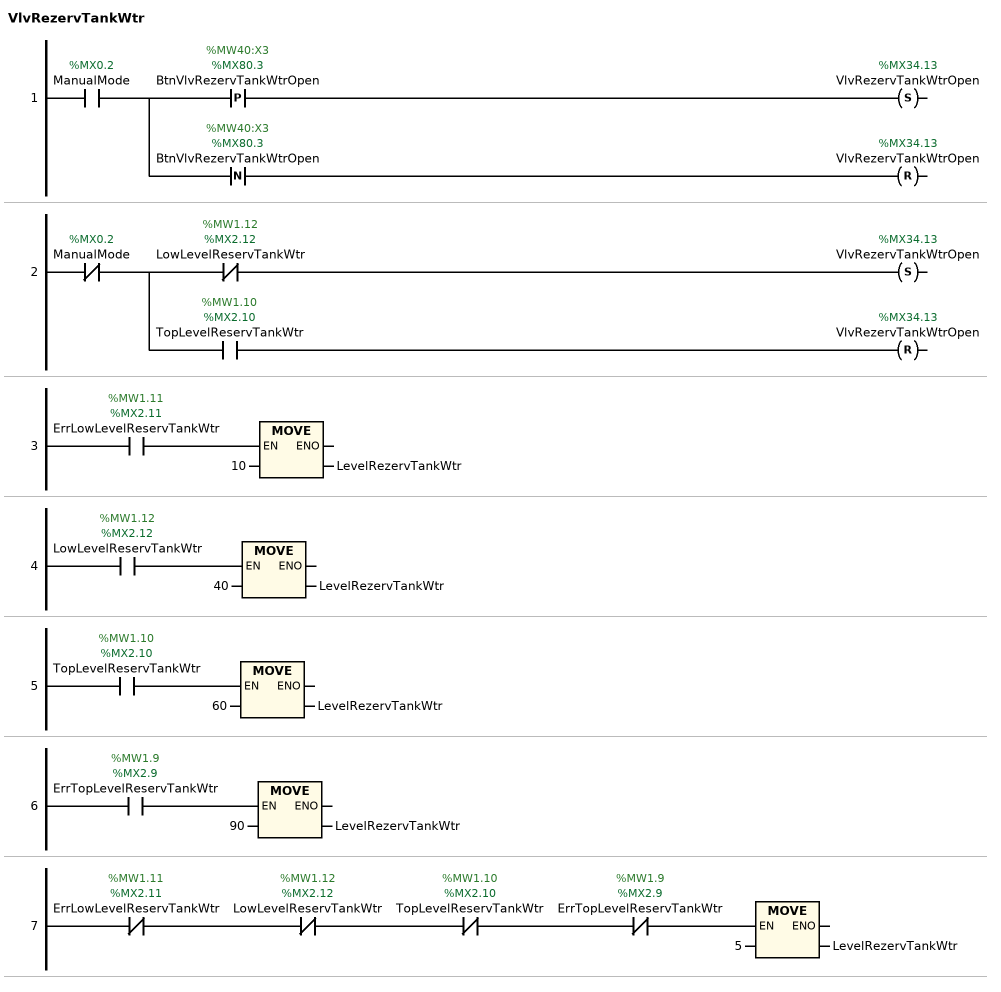
// NETWORK 1
//   ManualMode: AT %MX0.2
//   BtnVlvRezervTankWtrOpen: %MW40:X3 | AT %MX80.3
//   VlvRezervTankWtrOpen: AT %MX34.13
_rt1(CLK := BtnVlvRezervTankWtrOpen);
VlvRezervTankWtrOpen S= ManualMode AND _rt1.Q;
_ft1(CLK := BtnVlvRezervTankWtrOpen);
VlvRezervTankWtrOpen R= ManualMode AND _ft1.Q;

// NETWORK 2
//   ManualMode: AT %MX0.2
//   LowLevelReservTankWtr: %MW1.12 | AT %MX2.12
//   VlvRezervTankWtrOpen: AT %MX34.13
//   TopLevelReservTankWtr: %MW1.10 | AT %MX2.10
_w1 := NOT ManualMode;
VlvRezervTankWtrOpen S= _w1 AND NOT LowLevelReservTankWtr;
VlvRezervTankWtrOpen R= _w1 AND TopLevelReservTankWtr;

// NETWORK 3
//   ErrLowLevelReservTankWtr: %MW1.11 | AT %MX2.11
//   LevelRezervTankWtr: AT %MW41
IF ErrLowLevelReservTankWtr THEN LevelRezervTankWtr := 10; END_IF

// NETWORK 4
//   LowLevelReservTankWtr: %MW1.12 | AT %MX2.12
//   LevelRezervTankWtr: AT %MW41
IF LowLevelReservTankWtr THEN LevelRezervTankWtr := 40; END_IF

// NETWORK 5
//   TopLevelReservTankWtr: %MW1.10 | AT %MX2.10
//   LevelRezervTankWtr: AT %MW41
IF TopLevelReservTankWtr THEN LevelRezervTankWtr := 60; END_IF

// NETWORK 6
//   ErrTopLevelReservTankWtr: %MW1.9 | AT %MX2.9
//   LevelRezervTankWtr: AT %MW41
IF ErrTopLevelReservTankWtr THEN LevelRezervTankWtr := 90; END_IF

// NETWORK 7
//   ErrLowLevelReservTankWtr: %MW1.11 | AT %MX2.11
//   LowLevelReservTankWtr: %MW1.12 | AT %MX2.12
//   TopLevelReservTankWtr: %MW1.10 | AT %MX2.10
//   ErrTopLevelReservTankWtr: %MW1.9 | AT %MX2.9
//   LevelRezervTankWtr: AT %MW41
IF NOT ErrLowLevelReservTankWtr AND NOT LowLevelReservTankWtr AND NOT TopLevelReservTankWtr AND NOT ErrTopLevelReservTankWtr THEN
    LevelRezervTankWtr := 5;
END_IF

END_PROGRAM

// MyController/Application/PRG/SetResetErr
PROGRAM SetResetErr
VAR
	RunSignal: BLINK;
	tp_reset: TP;
	TpResetErr: TP;
	TonResetErr: TON;
END_VAR

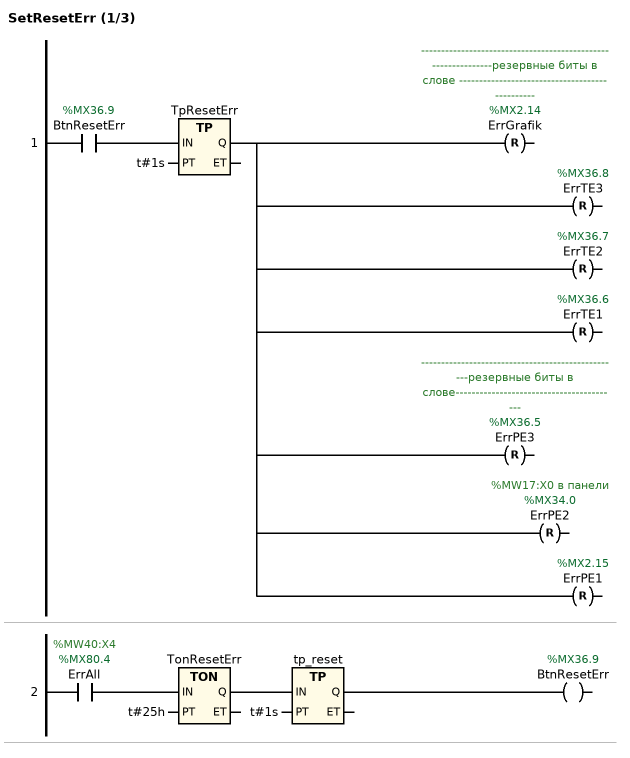
// NETWORK 1
//   BtnResetErr: AT %MX36.9
//   ErrGrafik: --------------------------------------------------------------резервные биты в слове ----------------------------------------------- | AT %MX2.14
//   ErrTE3: AT %MX36.8
//   ErrTE2: AT %MX36.7
//   ErrTE1: AT %MX36.6
//   ErrPE3: --------------------------------------------------резервные биты в слове----------------------------------------- | AT %MX36.5
//   ErrPE2: %MW17:X0 в панели | AT %MX34.0
//   ErrPE1: AT %MX2.15
TpResetErr(IN := BtnResetErr, PT := t#1s); // TP
ErrGrafik R= TpResetErr.Q;
ErrTE3 R= TpResetErr.Q;
ErrTE2 R= TpResetErr.Q;
ErrTE1 R= TpResetErr.Q;
ErrPE3 R= TpResetErr.Q;
ErrPE2 R= TpResetErr.Q;
ErrPE1 R= TpResetErr.Q;

// NETWORK 2
//   ErrAll: %MW40:X4 | AT %MX80.4
//   BtnResetErr: AT %MX36.9
TonResetErr(IN := ErrAll, PT := t#25h); // TON
tp_reset(IN := TonResetErr.Q, PT := t#1s); // TP
BtnResetErr := tp_reset.Q;

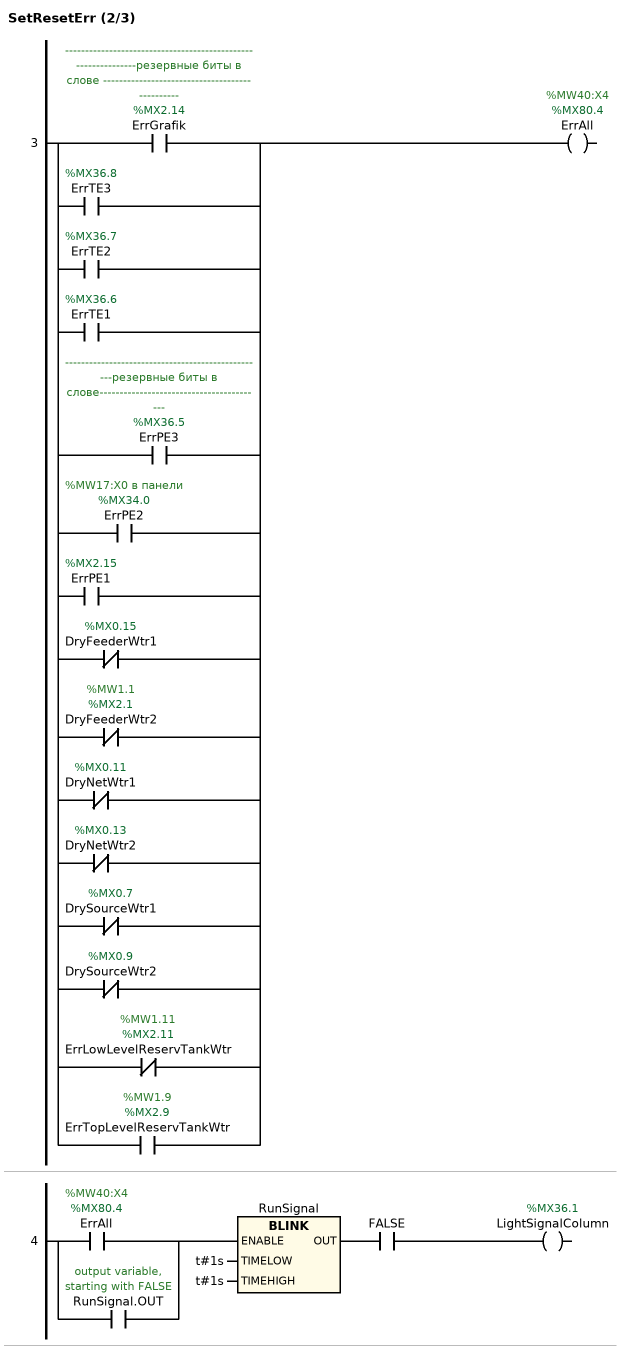
// NETWORK 3
//   ErrGrafik: --------------------------------------------------------------резервные биты в слове ----------------------------------------------- | AT %MX2.14
//   ErrTE3: AT %MX36.8
//   ErrTE2: AT %MX36.7
//   ErrTE1: AT %MX36.6
//   ErrPE3: --------------------------------------------------резервные биты в слове----------------------------------------- | AT %MX36.5
//   ErrPE2: %MW17:X0 в панели | AT %MX34.0
//   ErrPE1: AT %MX2.15
//   DryFeederWtr1: AT %MX0.15
//   DryFeederWtr2: %MW1.1 | AT %MX2.1
//   DryNetWtr1: AT %MX0.11
//   DryNetWtr2: AT %MX0.13
//   DrySourceWtr1: AT %MX0.7
//   DrySourceWtr2: AT %MX0.9
//   ErrLowLevelReservTankWtr: %MW1.11 | AT %MX2.11
//   ErrTopLevelReservTankWtr: %MW1.9 | AT %MX2.9
//   ErrAll: %MW40:X4 | AT %MX80.4
ErrAll := ErrGrafik OR ErrTE3 OR ErrTE2 OR ErrTE1 OR ErrPE3 OR ErrPE2 OR ErrPE1 OR NOT DryFeederWtr1 OR NOT DryFeederWtr2 OR NOT DryNetWtr1 OR NOT DryNetWtr2 OR NOT DrySourceWtr1 OR NOT DrySourceWtr2 OR NOT ErrLowLevelReservTankWtr OR ErrTopLevelReservTankWtr;

// NETWORK 4
//   ErrAll: %MW40:X4 | AT %MX80.4
//   RunSignal.OUT: output variable, starting with FALSE
//   LightSignalColumn: AT %MX36.1
RunSignal(ENABLE := ErrAll OR RunSignal.OUT, TIMELOW := t#1s, TIMEHIGH := t#1s); // BLINK
LightSignalColumn := RunSignal.OUT AND FALSE;

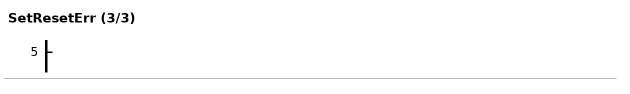
// NETWORK 5

END_PROGRAM

// MyController/Application/PRG/FactorySetup
PROGRAM FactorySetup
VAR
END_VAR
VAR // added by the converter: edge detectors and wires of the graphical bodies
    _rt1, _rt2, _rt3, _rt4, _rt5, _rt6, _rt7, _rt8, _rt9, _rt10, _rt11, _rt12, _rt13, _rt14, _rt15, _rt16, _rt17, _rt18, _rt19, _rt20, _rt21, _rt22, _rt23 : R_TRIG;
END_VAR

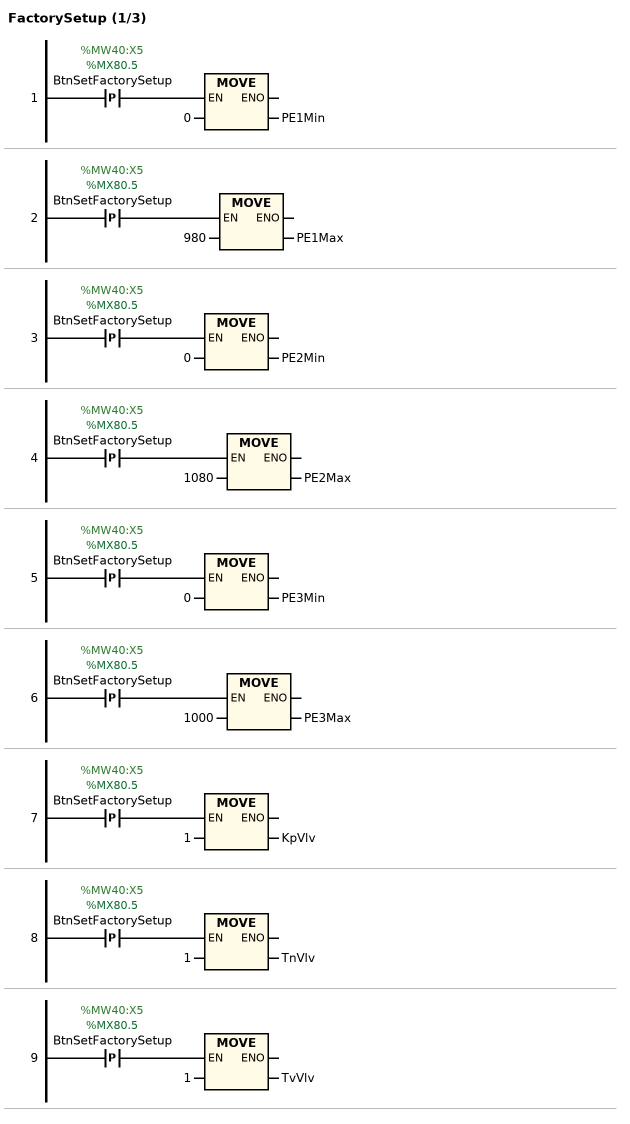
// NETWORK 1
//   BtnSetFactorySetup: %MW40:X5 | AT %MX80.5
//   PE1Min: AT %MW4
_rt1(CLK := BtnSetFactorySetup);
IF _rt1.Q THEN PE1Min := 0; END_IF

// NETWORK 2
//   BtnSetFactorySetup: %MW40:X5 | AT %MX80.5
//   PE1Max: AT %MW5
_rt2(CLK := BtnSetFactorySetup);
IF _rt2.Q THEN PE1Max := 980; END_IF

// NETWORK 3
//   BtnSetFactorySetup: %MW40:X5 | AT %MX80.5
//   PE2Min: AT %MW8
_rt3(CLK := BtnSetFactorySetup);
IF _rt3.Q THEN PE2Min := 0; END_IF

// NETWORK 4
//   BtnSetFactorySetup: %MW40:X5 | AT %MX80.5
//   PE2Max: AT %MW9
_rt4(CLK := BtnSetFactorySetup);
IF _rt4.Q THEN PE2Max := 1080; END_IF

// NETWORK 5
//   BtnSetFactorySetup: %MW40:X5 | AT %MX80.5
//   PE3Min: AT %MW12
_rt5(CLK := BtnSetFactorySetup);
IF _rt5.Q THEN PE3Min := 0; END_IF

// NETWORK 6
//   BtnSetFactorySetup: %MW40:X5 | AT %MX80.5
//   PE3Max: AT %MW13
_rt6(CLK := BtnSetFactorySetup);
IF _rt6.Q THEN PE3Max := 1000; END_IF

// NETWORK 7
//   BtnSetFactorySetup: %MW40:X5 | AT %MX80.5
//   KpVlv: %MW30, %MW31 | AT %MD15
_rt7(CLK := BtnSetFactorySetup);
IF _rt7.Q THEN KpVlv := 1; END_IF

// NETWORK 8
//   BtnSetFactorySetup: %MW40:X5 | AT %MX80.5
//   TnVlv: %MW32, %MW33 | AT %MD16
_rt8(CLK := BtnSetFactorySetup);
IF _rt8.Q THEN TnVlv := 1; END_IF

// NETWORK 9
//   BtnSetFactorySetup: %MW40:X5 | AT %MX80.5
//   TvVlv: %MW34, %MW35 | AT %MD17
_rt9(CLK := BtnSetFactorySetup);
IF _rt9.Q THEN TvVlv := 1; END_IF

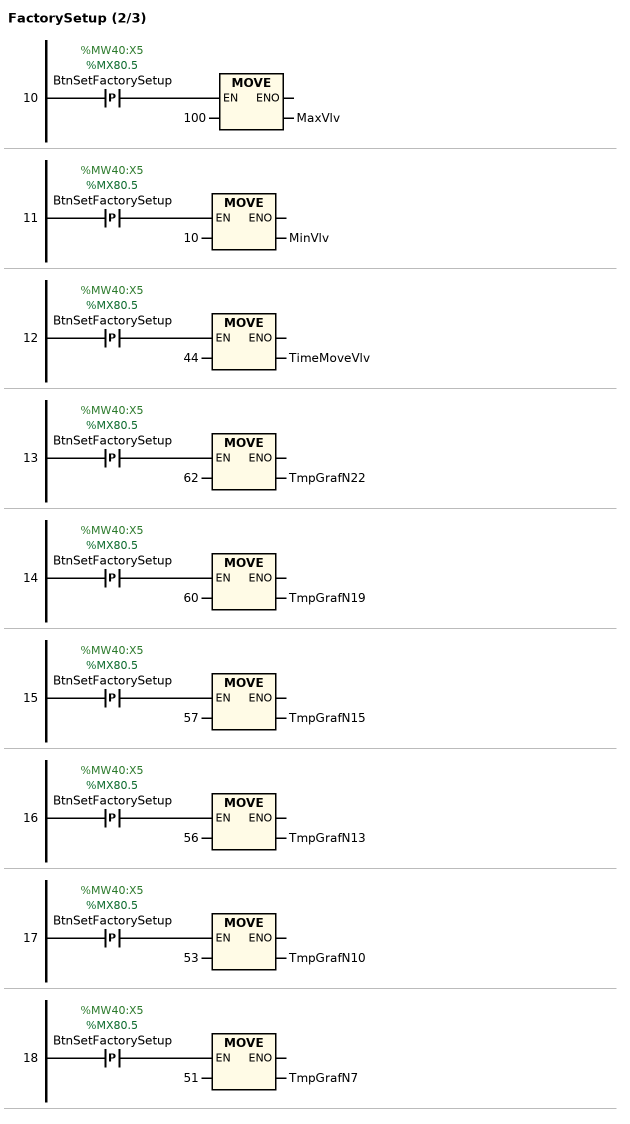
// NETWORK 10
//   BtnSetFactorySetup: %MW40:X5 | AT %MX80.5
//   MaxVlv: Максимальная величина открытия задвижки в % | AT %MW36
_rt10(CLK := BtnSetFactorySetup);
IF _rt10.Q THEN MaxVlv := 100; END_IF

// NETWORK 11
//   BtnSetFactorySetup: %MW40:X5 | AT %MX80.5
//   MinVlv: Минимальная величина закрытия задвижки в % | AT %MW37
_rt11(CLK := BtnSetFactorySetup);
IF _rt11.Q THEN MinVlv := 10; END_IF

// NETWORK 12
//   BtnSetFactorySetup: %MW40:X5 | AT %MX80.5
//   TimeMoveVlv: Время открытия задвижки в секундах | AT %MW38
_rt12(CLK := BtnSetFactorySetup);
IF _rt12.Q THEN TimeMoveVlv := 44; END_IF

// NETWORK 13
//   BtnSetFactorySetup: %MW40:X5 | AT %MX80.5
//   TmpGrafN22: AT %MW19
_rt13(CLK := BtnSetFactorySetup);
IF _rt13.Q THEN TmpGrafN22 := 62; END_IF

// NETWORK 14
//   BtnSetFactorySetup: %MW40:X5 | AT %MX80.5
//   TmpGrafN19: AT %MW20
_rt14(CLK := BtnSetFactorySetup);
IF _rt14.Q THEN TmpGrafN19 := 60; END_IF

// NETWORK 15
//   BtnSetFactorySetup: %MW40:X5 | AT %MX80.5
//   TmpGrafN15: AT %MW21
_rt15(CLK := BtnSetFactorySetup);
IF _rt15.Q THEN TmpGrafN15 := 57; END_IF

// NETWORK 16
//   BtnSetFactorySetup: %MW40:X5 | AT %MX80.5
//   TmpGrafN13: AT %MW22
_rt16(CLK := BtnSetFactorySetup);
IF _rt16.Q THEN TmpGrafN13 := 56; END_IF

// NETWORK 17
//   BtnSetFactorySetup: %MW40:X5 | AT %MX80.5
//   TmpGrafN10: AT %MW23
_rt17(CLK := BtnSetFactorySetup);
IF _rt17.Q THEN TmpGrafN10 := 53; END_IF

// NETWORK 18
//   BtnSetFactorySetup: %MW40:X5 | AT %MX80.5
//   TmpGrafN7: AT %MW24
_rt18(CLK := BtnSetFactorySetup);
IF _rt18.Q THEN TmpGrafN7 := 51; END_IF

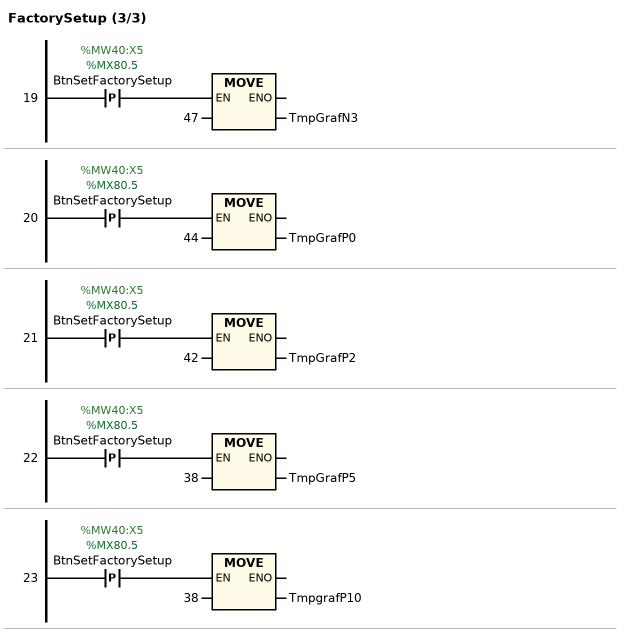
// NETWORK 19
//   BtnSetFactorySetup: %MW40:X5 | AT %MX80.5
//   TmpGrafN3: AT %MW25
_rt19(CLK := BtnSetFactorySetup);
IF _rt19.Q THEN TmpGrafN3 := 47; END_IF

// NETWORK 20
//   BtnSetFactorySetup: %MW40:X5 | AT %MX80.5
//   TmpGrafP0: AT %MW26
_rt20(CLK := BtnSetFactorySetup);
IF _rt20.Q THEN TmpGrafP0 := 44; END_IF

// NETWORK 21
//   BtnSetFactorySetup: %MW40:X5 | AT %MX80.5
//   TmpGrafP2: AT %MW27
_rt21(CLK := BtnSetFactorySetup);
IF _rt21.Q THEN TmpGrafP2 := 42; END_IF

// NETWORK 22
//   BtnSetFactorySetup: %MW40:X5 | AT %MX80.5
//   TmpGrafP5: AT %MW28
_rt22(CLK := BtnSetFactorySetup);
IF _rt22.Q THEN TmpGrafP5 := 38; END_IF

// NETWORK 23
//   BtnSetFactorySetup: %MW40:X5 | AT %MX80.5
//   TmpgrafP10: AT %MW29
_rt23(CLK := BtnSetFactorySetup);
IF _rt23.Q THEN TmpgrafP10 := 38; END_IF

END_PROGRAM

// MyController/Application/PRG/PumpsSourceWater
PROGRAM PumpsSourceWater
VAR
	PulsRunPumpSourceWtr1: TP;
	PulsStopPumpSourceWtr1: TP;
	PulsStopPumpSourceWtr2: TP;
	PulsRunPumpSourceWtr2: TP;
END_VAR
VAR // added by the converter: edge detectors and wires of the graphical bodies
    _w1 : BOOL;
    _rt1, _rt2, _rt3, _rt4 : R_TRIG;
    _ft1, _ft2 : F_TRIG;
END_VAR

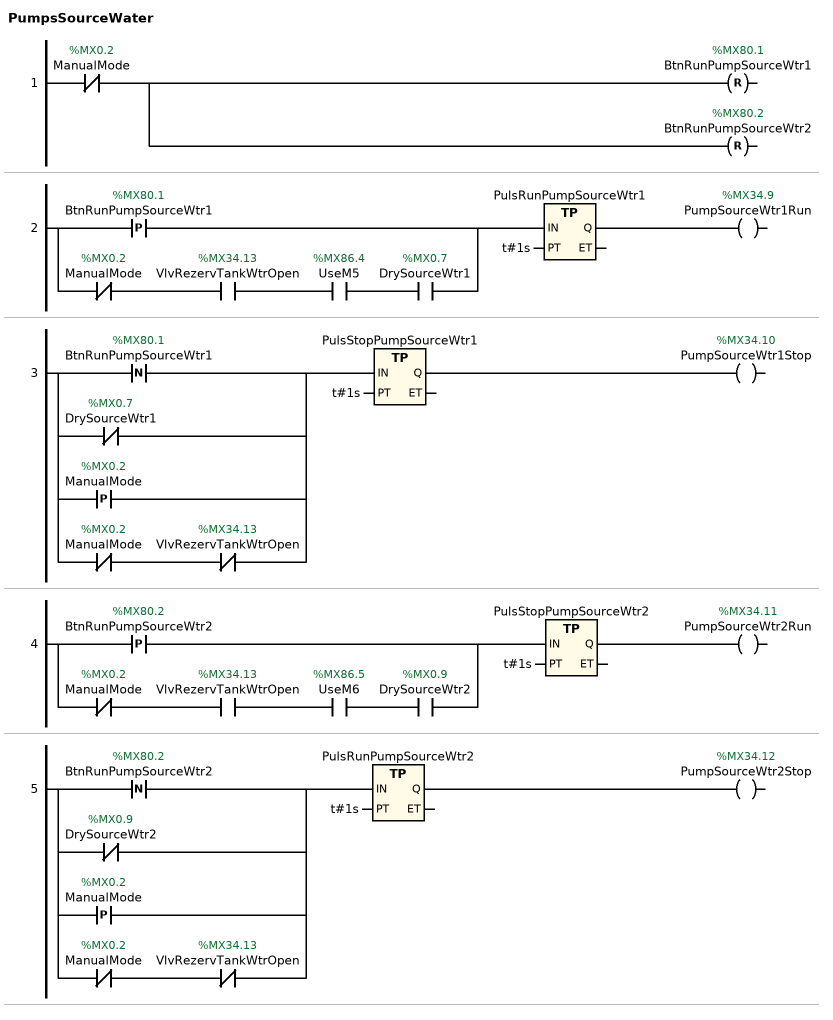
// NETWORK 1
//   ManualMode: AT %MX0.2
//   BtnRunPumpSourceWtr1: AT %MX80.1
//   BtnRunPumpSourceWtr2: AT %MX80.2
_w1 := NOT ManualMode;
BtnRunPumpSourceWtr1 R= _w1;
BtnRunPumpSourceWtr2 R= _w1;

// NETWORK 2
//   BtnRunPumpSourceWtr1: AT %MX80.1
//   ManualMode: AT %MX0.2
//   VlvRezervTankWtrOpen: AT %MX34.13
//   UseM5: AT %MX86.4
//   DrySourceWtr1: AT %MX0.7
//   PumpSourceWtr1Run: AT %MX34.9
_rt1(CLK := BtnRunPumpSourceWtr1);
PulsRunPumpSourceWtr1(IN := _rt1.Q OR NOT ManualMode AND VlvRezervTankWtrOpen AND UseM5 AND DrySourceWtr1, PT := t#1s); // TP
PumpSourceWtr1Run := PulsRunPumpSourceWtr1.Q;

// NETWORK 3
//   BtnRunPumpSourceWtr1: AT %MX80.1
//   DrySourceWtr1: AT %MX0.7
//   ManualMode: AT %MX0.2
//   VlvRezervTankWtrOpen: AT %MX34.13
//   PumpSourceWtr1Stop: AT %MX34.10
_ft1(CLK := BtnRunPumpSourceWtr1);
_rt2(CLK := ManualMode);
PulsStopPumpSourceWtr1(IN := _ft1.Q OR NOT DrySourceWtr1 OR _rt2.Q OR NOT ManualMode AND NOT VlvRezervTankWtrOpen, PT := t#1s); // TP
PumpSourceWtr1Stop := PulsStopPumpSourceWtr1.Q;

// NETWORK 4
//   BtnRunPumpSourceWtr2: AT %MX80.2
//   ManualMode: AT %MX0.2
//   VlvRezervTankWtrOpen: AT %MX34.13
//   UseM6: AT %MX86.5
//   DrySourceWtr2: AT %MX0.9
//   PumpSourceWtr2Run: AT %MX34.11
_rt3(CLK := BtnRunPumpSourceWtr2);
PulsStopPumpSourceWtr2(IN := _rt3.Q OR NOT ManualMode AND VlvRezervTankWtrOpen AND UseM6 AND DrySourceWtr2, PT := t#1s); // TP
PumpSourceWtr2Run := PulsStopPumpSourceWtr2.Q;

// NETWORK 5
//   BtnRunPumpSourceWtr2: AT %MX80.2
//   DrySourceWtr2: AT %MX0.9
//   ManualMode: AT %MX0.2
//   VlvRezervTankWtrOpen: AT %MX34.13
//   PumpSourceWtr2Stop: AT %MX34.12
_ft2(CLK := BtnRunPumpSourceWtr2);
_rt4(CLK := ManualMode);
PulsRunPumpSourceWtr2(IN := _ft2.Q OR NOT DrySourceWtr2 OR _rt4.Q OR NOT ManualMode AND NOT VlvRezervTankWtrOpen, PT := t#1s); // TP
PumpSourceWtr2Stop := PulsRunPumpSourceWtr2.Q;

END_PROGRAM

// MyController/Application/PRG/PumpsNetWater
PROGRAM PumpsNetWater
VAR
	PulsRunPumpNetWtr1: TP;
	PulsStopPumpNetWtr1: TP;
	PulsStopPumpNetWtr2: TP;
	PulsRunPumpNetWtr2: TP;
END_VAR
VAR // added by the converter: edge detectors and wires of the graphical bodies
    _w1 : BOOL;
    _rt1, _rt2, _rt3, _rt4 : R_TRIG;
    _ft1, _ft2 : F_TRIG;
END_VAR

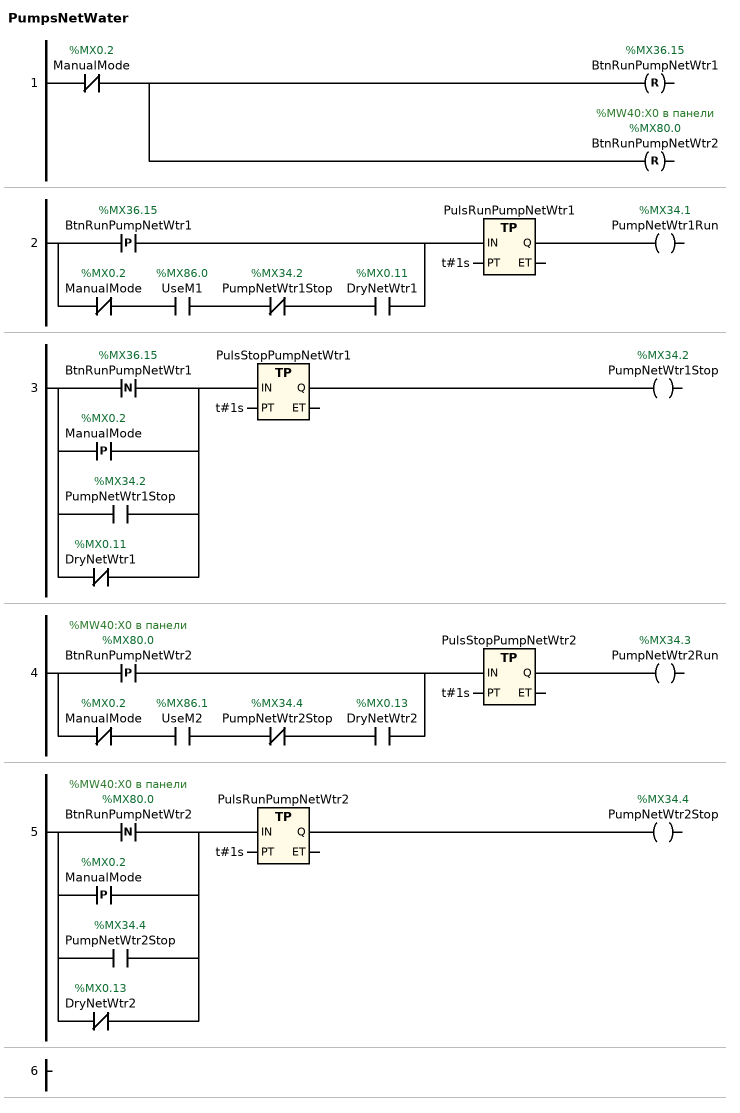
// NETWORK 1
//   ManualMode: AT %MX0.2
//   BtnRunPumpNetWtr1: AT %MX36.15
//   BtnRunPumpNetWtr2: %MW40:X0 в панели | AT %MX80.0
_w1 := NOT ManualMode;
BtnRunPumpNetWtr1 R= _w1;
BtnRunPumpNetWtr2 R= _w1;

// NETWORK 2
//   BtnRunPumpNetWtr1: AT %MX36.15
//   ManualMode: AT %MX0.2
//   UseM1: AT %MX86.0
//   PumpNetWtr1Stop: AT %MX34.2
//   DryNetWtr1: AT %MX0.11
//   PumpNetWtr1Run: AT %MX34.1
_rt1(CLK := BtnRunPumpNetWtr1);
PulsRunPumpNetWtr1(IN := _rt1.Q OR NOT ManualMode AND UseM1 AND NOT PumpNetWtr1Stop AND DryNetWtr1, PT := t#1s); // TP
PumpNetWtr1Run := PulsRunPumpNetWtr1.Q;

// NETWORK 3
//   BtnRunPumpNetWtr1: AT %MX36.15
//   ManualMode: AT %MX0.2
//   PumpNetWtr1Stop: AT %MX34.2
//   DryNetWtr1: AT %MX0.11
_ft1(CLK := BtnRunPumpNetWtr1);
_rt2(CLK := ManualMode);
PulsStopPumpNetWtr1(IN := _ft1.Q OR _rt2.Q OR PumpNetWtr1Stop OR NOT DryNetWtr1, PT := t#1s); // TP
PumpNetWtr1Stop := PulsStopPumpNetWtr1.Q;

// NETWORK 4
//   BtnRunPumpNetWtr2: %MW40:X0 в панели | AT %MX80.0
//   ManualMode: AT %MX0.2
//   UseM2: AT %MX86.1
//   PumpNetWtr2Stop: AT %MX34.4
//   DryNetWtr2: AT %MX0.13
//   PumpNetWtr2Run: AT %MX34.3
_rt3(CLK := BtnRunPumpNetWtr2);
PulsStopPumpNetWtr2(IN := _rt3.Q OR NOT ManualMode AND UseM2 AND NOT PumpNetWtr2Stop AND DryNetWtr2, PT := t#1s); // TP
PumpNetWtr2Run := PulsStopPumpNetWtr2.Q;

// NETWORK 5
//   BtnRunPumpNetWtr2: %MW40:X0 в панели | AT %MX80.0
//   ManualMode: AT %MX0.2
//   PumpNetWtr2Stop: AT %MX34.4
//   DryNetWtr2: AT %MX0.13
_ft2(CLK := BtnRunPumpNetWtr2);
_rt4(CLK := ManualMode);
PulsRunPumpNetWtr2(IN := _ft2.Q OR _rt4.Q OR PumpNetWtr2Stop OR NOT DryNetWtr2, PT := t#1s); // TP
PumpNetWtr2Stop := PulsRunPumpNetWtr2.Q;

// NETWORK 6

END_PROGRAM

// MyController/Application/FB/ControlMeteoVlv
FUNCTION_BLOCK ControlMeteoVlv
VAR_INPUT
	TARGET: REAL;
END_VAR
VAR_OUTPUT
	OPEN: BOOL;
	CLOSE: BOOL;
END_VAR
VAR
	PulsValveOpn: BLINK;
	PulsValveClose: BLINK;
END_VAR

//Импульсно открываем задвижку
PulsValveOpn.TIMEHIGH := T#1S;
PulsValveOpn.TIMELOW := T#5S;
PulsValveOpn.ENABLE := ((TARGET>CurrentPosition AND NOT HandModeMeteo) OR PulsValveOpn.OUT);
OPEN := PulsValveOpn.OUT;

//Импульсно закрываем задвижку
PulsValveClose.TIMEHIGH := T#1S;
PulsValveClose.TIMELOW := T#5S;
PulsValveClose.ENABLE := ((TARGET<CurrentPosition AND NOT HandModeMeteo) OR PulsValveClose.OUT);
CLOSE := PulsValveClose.OUT;

END_FUNCTION_BLOCK

// MyController/Application/CheckDivDInt
// Implicitly generated code : DO NOT EDIT
FUNCTION CheckDivDInt : DINT
VAR_INPUT
	divisor:DINT;
END_VAR

// Implicitly generated code : Only an Implementation suggestion
IF divisor = 0 THEN
	CheckDivDInt:=1;
ELSE
	CheckDivDInt:=divisor;
END_IF;

END_FUNCTION

// MyController/Application/CheckDivLInt
// Implicitly generated code : DO NOT EDIT
FUNCTION CheckDivLInt : LINT
VAR_INPUT
	divisor:LINT;
END_VAR

// Implicitly generated code : Only an Implementation suggestion
IF divisor = 0 THEN
	CheckDivLInt:=1;
ELSE
	CheckDivLInt:=divisor;
END_IF;

END_FUNCTION

// MyController/Application/CheckDivLReal
// Implicitly generated code : DO NOT EDIT
FUNCTION CheckDivLReal : LREAL
VAR_INPUT
	divisor:LREAL;
END_VAR

// Implicitly generated code : Only an Implementation suggestion
IF divisor = 0 THEN
	CheckDivLReal:=1;
ELSE
	CheckDivLReal:=divisor;
END_IF;

END_FUNCTION
